Staubli VAL3: userPage.pjx

--- userPage.pjx ---
Parameters version=s7.3.1 stackSize=5000 millimeterUnit=true
Program file=changeValue.pgx
Program file=clear.pgx
Program file=CompareStrArray.pgx
Program file=divideString.pgx
Program file=editNum.pgx
Program file=editNumField.pgx
Program file=editNumField1.pgx
Program file=editStr.pgx
Program file=example.pgx
Program file=findPos.pgx
Program file=getListPosition.pgx
Program file=getMenu.pgx
Program file=getView.pgx
Program file=insertDialog.pgx
Program file=isListEmpty.pgx
Program file=leftPos.pgx
Program file=listadd.pgx
Program file=listcreate.pgx
Program file=listcursor.pgx
Program file=listdel.pgx
Program file=listempty.pgx
Program file=listevent.pgx
Program file=listframe.pgx
Program file=listins.pgx
Program file=listredraw.pgx
Program file=listupdate.pgx
Program file=listupdate1.pgx
Program file=midPos.pgx
Program file=nullKey.pgx
Program file=numCopy.pgx
Program file=printScroll.pgx
Program file=questionDialog.pgx
Program file=read.pgx
Program file=rightPos.pgx
Program file=scroll.pgx
Program file=selectNewField.pgx
Program file=setCenter.pgx
Program file=setList.pgx
Program file=setMenu.pgx
Program file=SetProerty.pgx
Program file=setSizeList.pgx
Program file=setView.pgx
Program file=showBoolStatus.pgx
Program file=strfill.pgx
Program file=strfillchr.pgx
Program file=stringCopy.pgx
Program file=stringToArray.pgx
Program file=strlength.pgx
Program file=timerDialog.pgx
Program file=type.pgx
Program file=typeCenter.pgx
Program file=typeLen.pgx
Program file=typeMenu.pgx
Program file=yes.pgx
Program file=yes_no.pgx
Program file=yes_no_cancel.pgx
Data file=userPage.dtx

--- changeValue.pgx ---
public program changeValue(num& x_nValue[], num x_nMin, num x_nMax, num x_nX, num x_nY, string& x_sItem[])
  local num l_nOldValue[2]
  local string l_sItem
  local string l_sMessage
  local bool l_bComma
  local string l_sEmpty
begin
  //-----------------------------------------------------------------------
  //Header begin
  //Description of program
  //  Get a numerical value on the x_nX column and x_nY line and test if
  //  the value is between x_nMin and x_nMax. If the two parameters x_nMin
  //  and x_nMax are equal there are no limits.
  //  If x_sItems is not Empty, the program displays the list of Items and
  //  you can change the selected Item : the index is returned in x_nValue.
  //
  //Input parameters
  //  num x_nMin :
  //    role : min value limit
  //  num x_nMax :
  //    role : max value limit
  //  num x_nX :
  //    role : X cursor position for change the value
  //  num x_nY :
  //    role : Y cursor position for change the value
  //
  //Output paramaters
  //  num x_nValue :
  //    role : numerical value changed or index pointer of x_sItem
  //  string x_sItems
  //    role : array of Items
  //
  //Example
  //  call changeValue(l_nValue,0,10,2,5,"") //The user can changed the numerical
  //                                           value of l_nValue. If the seized
  //                                           is not between 0 to 10 the user must
  //                                           changed the value.
  //
  //  call changeValue(l_nValue,0,10,2,5,sItem) //The list sItem is displaying on
  //                                              the screen and the user select one
  //                                              element of the list. The index
  //                                              is returned in l_nValue.
  //
  //
  //History
  //  Creation : 28-04-08 - f.Rob
  //Header end
  //-----------------------------------------------------------------------

  if x_nMin>x_nMax
    return
  endIf
  //Print the line in white
  call nullKey(nKey)
  l_nOldValue[1]=round(x_nValue)
  x_nValue=(round(x_nValue*100))/100
  l_nOldValue=x_nValue
  //Check if is using the comma or not
  if l_nOldValue!=l_nOldValue[1]
    l_bComma=true
  else
    l_bComma=false
  endIf
  //Start
  do
    if x_sItem==""
      //Use the get num
      if l_bComma
        call strfill(l_sEmpty,len(toString("8.3",x_nValue)),l_sEmpty)
      else
        call strfill(l_sEmpty,len(toString("8.3",x_nValue)),l_sEmpty)
      endIf
      call type(x_nX,x_nY,l_sEmpty)
      gotoxy(x_nX,x_nY)
      nKey=get(x_nValue)
      // CHECK for MIN MAX VALUE
      if x_nMax!=x_nMin
        if x_nValue>x_nMax
          //Ask if you want to continue
          popUpMsg("MAX: "+toString(".2",x_nMax))
          x_nValue=l_nOldValue
          //x_nValue=x_nMax
          nKey=-1
        else
          if x_nValue<x_nMin
            popUpMsg("MIN: "+toString(".2",x_nMin))
            //x_nValue=x_nMin
            x_nValue=l_nOldValue
            nKey=-1
          endIf
        endIf
      endIf
      // UPDATE THE VALUE
      if l_bComma
        call type(x_nX,x_nY,toString("8.3",x_nValue))
      else
        call type(x_nX,x_nY,toString("8.3",x_nValue))
      endIf
    else
//      // STRING CHOICE
//      nKey=getKey()
//      switch nKey
//        // CHANGE THE ITEMS ARRAY
//        case 261
//          // UP
//          x_nValue=abs((x_nValue+1)%size(x_sItem))
//        break
//        case 266
//          // DOWN
//          x_nValue=abs((x_nValue+size(x_sItem)-1)%size(x_sItem))
//        break
//      endSwitch
//      // UPDATE THE VALUE
//      setTextMode(3)
//      call typeLen(x_nX,x_nY,x_sItem[x_nValue],8)
//      setTextMode(0)
    endIf
    //Release the resource
    delay(0)
  until nKey==270 or nKey==255
  if nKey==255
    bUseEscape=true
    x_nValue=l_nOldValue
//    if x_sItem!=""
//      x_sItem=x_sItem[l_nOldValue]
//    endIf
  else
    bUseEscape=false
  endIf
  //Leave the resource
  delay(0)
end

--- divideString.pgx ---
program divideString(string& x_sMsg[] (dimensions=1), num& x_nLine[] (dimensions=1))
  local string l_sCopyMsg
  local num l_nLength
  local string l_sSwap
  local num l_nFlag
  local num l_nTotalFlag
  local string l_sCR
  local num l_nPosCR
  local num i
begin
  //
  //  using:
  // x_sMessage->  the message you want print to video
  // x_nLine->     the number of the line that will be use
  //
  //
  // CARRIAGE RETURN
  l_sCR="#"
  x_nLine=0
  //length of a line for a message
  l_nLength=38
  // copy the msg
  l_sCopyMsg=x_sMsg
  // first case
  call findPos(l_sCopyMsg,l_sCR,l_nPosCR)
  if (getDisplayLen(l_sCopyMsg)>l_nLength-1) or (l_nPosCR!=-1)
    // compose the message
    do
      l_sSwap=l_sCopyMsg
      // set the x_sMsg
      if size(x_sMsg)-1<x_nLine
        append(x_sMsg)
      endIf
      call findPos(l_sCopyMsg,l_sCR,l_nPosCR)
      //
      if (getDisplayLen(l_sCopyMsg)>l_nLength-1 or (l_nPosCR!=-1)) and x_nLine<8
        // divide the string
        l_nTotalFlag=0
        call findPos(l_sCopyMsg,l_sCR,l_nPosCR)
        //
        // divide the string
        //
        if l_nPosCR!=-1 and l_nPosCR<l_nLength
          // CARRIAGE RETURN
          call leftPos(l_sCopyMsg,l_nPosCR,l_sSwap)
          //l_sSwap=left(l_sCopyMsg,l_nPosCR)
          call rightPos(l_sCopyMsg,getDisplayLen(l_sCopyMsg)-(l_nPosCR)-1,l_sCopyMsg)
          //l_sCopyMsg=right(l_sCopyMsg,len(l_sCopyMsg)-(l_nPosCR)-1)
          if getDisplayLen(l_sSwap)==0
            l_sSwap=" "
          endIf
        else
          //
          // search for the space then return
          //
          do
            call findPos(l_sSwap," ",l_nFlag)
            //l_nFlag=find(l_sSwap," ")
            if l_nFlag!=-1 and l_nFlag<=l_nLength
              //l_sSwap=right(l_sSwap,len(l_sSwap)-l_nFlag-1)
              call rightPos(l_sSwap,getDisplayLen(l_sSwap)-l_nFlag-1,l_sSwap)
              l_nTotalFlag=l_nTotalFlag+l_nFlag+1
            else
              if l_nTotalFlag==0 and (l_nFlag==-1 or l_nFlag>l_nLength)
                l_nFlag=-1
                l_nTotalFlag=38
              endIf
            endIf
          until l_nTotalFlag>=l_nLength+2 or l_nFlag==-1
          // NORMAL
          if l_nTotalFlag==0
            // FULL LINE
            call leftPos(l_sCopyMsg,l_nLength,l_sSwap)
            //l_sSwap=left(l_sCopyMsg,l_nLength)
            //l_sCopyMsg=right(l_sCopyMsg,len(l_sCopyMsg)-l_nLength)
            call rightPos(l_sCopyMsg,getDisplayLen(l_sCopyMsg)-l_nLength,l_sCopyMsg)
          else
            // DIVIDE IT
            call leftPos(l_sCopyMsg,l_nTotalFlag-l_nFlag-2,l_sSwap)
            //l_sSwap=left(l_sCopyMsg,l_nTotalFlag-l_nFlag-2)
            //l_sCopyMsg=right(l_sCopyMsg,len(l_sCopyMsg)-(l_nTotalFlag-l_nFlag-1))
            call rightPos(l_sCopyMsg,getDisplayLen(l_sCopyMsg)-(l_nTotalFlag-l_nFlag-1),l_sCopyMsg)
          endIf
        endIf
        // set the string
        x_sMsg[x_nLine]=l_sSwap
        x_nLine=x_nLine+1
      else
        // limit the string
        call rightPos(l_sSwap,l_nLength,x_sMsg[x_nLine])
        //x_sMsg[x_nLine]=right(l_sSwap,l_nLength)
        l_sSwap=""
      endIf
    until l_sSwap==""
  endIf
end

--- getView.pgx ---
public program getView(bool& x_bView[] (dimensions=1))
begin
  if nBottomX==38
    x_bView=true
  else
    x_bView=false
  endIf
end

--- insertDialog.pgx ---
public program insertDialog(string x_sMsg, num& x_nItem[], num x_nMin, num x_nMax)
  local num l_nStartLine
  local num l_nLine
  local num i
  local num l_nPX
  local num l_nPY
  local string l_sItem
  local string l_sMessage
  local string l_sEmpty
begin
  //
  // modify the x_sItem, using a min max range
  //
  if watch(bShowDialog==false,2)==false
    bShowDialog=false
    logMsg("error dialog resoursing")
    return
  else
    setMutex(bShowDialog)
    // clear the line
    call clear(0,13)
    // look for the comma
    if round(x_nItem)!=x_nItem
      l_sItem=toString(".2",x_nItem)
    else
      l_sItem=toString("",x_nItem)
    endIf
    // print the line
    l_sItem=x_sMsg+">"+l_sItem
    call stringCopy(l_sItem,sMessage)
    // divide the sentence
    call divideString(sMessage,l_nLine)
    l_nStartLine=round(5-l_nLine/2)
    // Start LINE
    call type(0,l_nStartLine-2,"┌──────────────────────────────────────┐")
    call type(0,l_nStartLine-1,"│                                      │")
    // write the message
    for i=0 to l_nLine
      //call type(,"                                      ")
      l_sMessage=sMessage[i]
      call typeCenter(i+l_nStartLine,l_sMessage,38,false)
      call type(0,l_nStartLine+i,"│"+l_sMessage+"│")
    endFor
    // end LINE
    call type(0,l_nStartLine+l_nLine+1,"│                                      │")
    call type(0,l_nStartLine+l_nLine+2,"└──────────────────────────────────────┘")
    l_nPX=find(l_sMessage,">")+2
    l_nPY=l_nStartLine+l_nLine
    // change the value
    call changeValue(x_nItem,x_nMin,x_nMax,l_nPX,l_nPY,l_sEmpty)
    //
    bShowDialog=false
    bUseRefresh=true
    //
    delay(0)
  endIf
end

--- listadd.pgx ---
public program listadd(string& x_sItems[] (dimensions=1))
  local num i
  local num l_nSize
begin
  //---------------------------------
  // insert x_sItems into the list
  //---------------------------------
  //
  // x_sItems:      Items to add
  //
  //---------------------------------
  // Staubli copyright 2005
  //                By toneage
  //[Public]-------------------------
  //
  //
  for i=0 to (size(x_sItems)-1)
    if (size(sItems)!=1 or sItems!="") and x_sItems[i]!=""
      insert(sItems[size(sItems)])
      insert(bReadWrite[size(bReadWrite)])
    endIf
    if x_sItems[i]!=""
      sItems[size(sItems)-1]=x_sItems[i]
      // for default the RW is true
      bReadWrite[size(bReadWrite)-1]=true
    endIf
  endFor
end

--- listupdate.pgx ---
public program listupdate(num pFirst (dimensions=1))
  local num lI
  local num lLen
  local string lStr
  local string lStr2
  local num lValue
  local num lView
  local num lX
  local num lY
  local num l_nSize
  local bool l_bEmpty
begin
  //
  // insert into the box all the data
  //
  // to prevent a negative value
  if pFirst>=0
    nFirst=pFirst
  else
    nFirst=0
  endIf
  // save the coordinate
  lValue=nBottomY-1
  // check the overFlow
  l_nSize=size(sItems)-1
  if (nFirst+nView>l_nSize)
    // reset the value
    nFirst=nView=0
  endIf
  lI=0
  // check the unKnow poblem
  if l_nSize<lValue
    if nFirst!=0
      nView=nView+nFirst
      nFirst=0
    endIf
  endIf
  do
    lX=nTopX+1
    lY=nBottomY+lI-1
    lY=nTopY+lI+1
    lLen=nBottomX
    if ((lI+nFirst)<size(sItems))
      // print the item
      if (l_nSize>=0)
        lStr=mid(sItems[(lI+nFirst)],lLen,0)
      endIf
    else
      // print the blank line
      lStr="                                        "
    endIf
    // fill the line
    call strfill(lStr,lLen,lStr2)
    gotoxy(lX,lY)
    put(lStr2)
    lI=lI+1
  until (lI>lValue)
  // underlien the actual line
  call isListEmpty(l_bEmpty)
  if !l_bEmpty
    call listcursor(nView,true)
  else
    call listcursor(nView,false)
    nView=0
    nFirst=0
  endIf
  // print the scroll
  call printScroll()
  // leave the resourse
  delay(0)
end

--- numCopy.pgx ---
public program numCopy(num& x_nCopy[] (dimensions=1), num& x_nPaste[] (dimensions=1))
// Copy all the value from the x_nCopy to x_nPaste
  local num i
  local num l_nSize
begin
  // Copy all the value from the first element to the second one
  //
  // redim the Paste String ARRAY
  //
  l_nSize=size(x_nPaste)
  if size(x_nCopy)>size(x_nPaste)
    for i=l_nSize to (size(x_nCopy)-1)
      insert(x_nPaste[i])
    endFor
  else
    if size(x_nCopy)<size(x_nPaste)
      for i=size(x_nCopy) to l_nSize-1
        delete(x_nPaste[size(x_nCopy)])
      endFor
    endIf
  endIf
  // COPY ALL THE FIELD
  for i=0 to (size(x_nCopy)-1)
    x_nPaste[i]=x_nCopy[i]
  endFor
end

--- setCenter.pgx ---
program setCenter()
begin
end

--- stringToArray.pgx ---
public program stringToArray(string x_sString (dimensions=1), string& x_sArray[] (dimensions=1))
// copy one String into an ARRAY of String
  local num i
  local num l_nItem
  local string l_sChar
  local string l_sEmpty
begin
  // define the char use to divide the items
  // PRIORITY
  //  ^
  //  ;
  //  ,
  //
  if find(x_sString,"^")==-1
    if find(x_sString,";")==-1
      l_sChar=","
    else
      l_sChar=";"
    endIf
  else
    l_sChar="^"
  endIf
  // init the X_sArray
  l_sEmpty=""
  call stringCopy(l_sEmpty,x_sArray)
  l_nItem=0
  do
    // increase the ARRAY SIZE
    if l_nItem>0
      insert(x_sArray[l_nItem])
    endIf
    i=find(x_sString,l_sChar)
    // look if was found
    if i!=-1
      // PUT INSIDE THE ARRAY THE STRING
      x_sArray[l_nItem]=left(x_sString,i)
      x_sString=delete(x_sString,i+1,0)
    else
      // look if is empty or not
      if len(x_sString)>0
        x_sArray[l_nItem]=(x_sString)
      endIf
    endIf
    l_nItem=l_nItem+1
  until i==-1
end

--- timerDialog.pgx ---
public program timerDialog(string x_sMsg (dimensions=1), num x_nTime (dimensions=1))
  local num l_nTime
  local num l_nStartLine
  local num l_nLine
  local num i
  local string l_sMessage
begin
  //
  // use for other task
  //
  if watch(bShowDialog==false,2)==false
    bShowDialog=false
    logMsg("error dialog resoursing")
    return
  else
    setMutex(bShowDialog)
    //
    //call listempty()
    //
    l_nTime=clock()
    call stringCopy(x_sMsg,sMessage)
    call divideString(sMessage,l_nLine)
    l_nStartLine=round(5-l_nLine/2)
    do
      // Start LINE
      call type(0,l_nStartLine-2,"┌──────────────────────────────────────┐")
      call type(0,l_nStartLine-1,"│                                      │")
      // write the message
      for i=0 to l_nLine
        call type(0,l_nStartLine+i,"")
        call type(39,l_nStartLine+i,"")
        //call typeCenter(i+l_nStartLine,sMessage[i],38,false)
        l_sMessage=sMessage[i]
        call typeCenter(i+l_nStartLine,l_sMessage,38,false)
        call type(0,l_nStartLine+i,"│"+l_sMessage+"│")
      endFor
      // end LINE
      call type(0,l_nStartLine+l_nLine+1,"│                                      │")
      call type(0,l_nStartLine+l_nLine+2,"└──────────────────────────────────────┘")
      // release
      if x_nTime==0
        delay(0.1)
      else
        delay(0)
      endIf
    until (clock()-l_nTime)>=x_nTime
    //
    bShowDialog=false
    bUseRefresh=true
    delay(0)
  endIf
  // bLocking=false
end

--- type.pgx ---
public program type(num pX (dimensions=1), num pY (dimensions=1), string pStr (dimensions=1))
begin
  //---------------------------------
  //  S H O W   O N E   S T R I N G
  //---------------------------------
  // Display one string to pX column
  // and pY Line
  //
  gotoxy(pX,pY)
  put(pStr)
end

--- typeMenu.pgx ---
public program typeMenu(num pNumber (dimensions=1), string pStr (dimensions=1))
  local string lStr
  local string lStrEmpty
  local num lMaxLen
  local num lPosX
  local num lPosY
  local num lStep
  local num i
begin
  //---------------------------------
  //  S H O W   O N E   S T R I N G
  //---------------------------------
  // Display one message in the
  // user menu page
  // 4 characters and 1 space
  //
  //
  lStep=5
  lPosY=13
  lStrEmpty="     "
  if (pNumber>=1) and (pNumber<=8)
    lMaxLen=4
    // Control the len
    // europe case
    if (getDisplayLen(pStr)>lMaxLen)
      if len(pStr)==getDisplayLen(pStr)
        i=find(pStr," ")
        if i<5 and i>2
          lStr=mid(pStr,i,0)
        else
          lStr=mid(pStr,lMaxLen-1,0)
          lStr=lStr+"."
        endIf
      else
        // asia one
        lStr=mid(pStr,2,0)
      endIf
    else
      lStr=pStr
    endIf
    // Position X
    lPosX=(pNumber-1)*lStep+1
    // log
    call strfill(lStr,4,lStr)
    call type(lPosX,lPosY,lStr)
  endIf
end

--- yes_no_cancel.pgx ---
public program yes_no_cancel(string x_sMessage (dimensions=1), string& x_sYesNo[] (dimensions=1), bool& x_bResult[] (dimensions=1), bool& x_bCancel[] (dimensions=1))
  local num i
  local string l_sButton[3]
begin
  // INIT
  x_bCancel=false
  l_sButton[0]=x_sYesNo
  l_sButton[1]=x_sYesNo[1]
  l_sButton[2]="Esc"
  // write a yes no cancel question dialog
  call questionDialog(x_sMessage,l_sButton,i)
  // press F8 or enter
  if i==1 or i==0
    x_bResult=true
  else
    // press escape or F6
    if i==-1 or i==3
      x_bCancel=true
    endIf
    // press F7-no
    x_bResult=false
  endIf
end
